(*
SPDX-FileCopyrightText: © 2026 Oleksandr Tiutyk <trofimich@gmail.com>
SPDX-License-Identifier: MIT
License: https://opensource.org/license/mit
*)

(*!
<summary>Reports a rejected filesystem path and its diagnostic explanation.</summary>
<description>
Reports caller-detected path errors using the GeneralException lifetime and throw rules. The path is borrowed
during the call; errorMessage is copied by value. Dynamic copies are explicitly registered by Clone after
construction; plain __NEW does not transfer ownership to the task manager.
</description>
*)

{attribute 'enable_dynamic_creation'}
{attribute 'no_explicit_call' := 'do not call this function block directly'}
FUNCTION_BLOCK InvalidPathException EXTENDS TOF_Core.GeneralException IMPLEMENTS IInvalidPathException
VAR_STAT
	//! <summary>Class name shared by all instances of this function block.</summary>
	{attribute 'hide'} 
	_ClassName : STRING := __POUNAME();
END_VAR

(*!
<summary>Provides the concrete type name used in diagnostics.</summary>
<description>
Returns borrowed read-only metadata; keep the instance alive and do not modify the referenced string.
Reading does not allocate memory, initialize resources or transfer ownership.
</description>
*)
{attribute 'monitoring' := 'call'}
PROPERTY ClassName : REFERENCE TO STRING
GET
ClassName REF= _ClassName;
END_GET
END_PROPERTY

(*!
<summary>Creates a task-owned copy of this exception and its diagnostic payload.</summary>
<description>
Registers the newly constructed instance before copying payload, outside FB_init. Registration failure
releases the unregistered instance and raises a terminal error; copy failure leaves the registered instance
owned by the task manager for cleanup. Custom overrides must follow the same ownership sequence. The returned
reference is borrowed until task cleanup and must not be deleted by the caller.
</description>
*)
METHOD Clone : TOF_Core.IObject
VAR
	exceptionClone : POINTER TO InvalidPathException;
END_VAR
exceptionClone := __NEW(InvalidPathException);

IF exceptionClone = 0 THEN
	TOF_Core.DynamicMemoryManager.RaiseAllocationFailure();
END_IF

TOF_Core.DynamicMemoryManager.RegisterAutoDisposedObject(autoDisposedObject := exceptionClone^);

exceptionClone^.CopyGeneralFields(sourceException := THIS^);

Clone := exceptionClone^;
END_METHOD

(*!
<summary>Provides the library namespace used in diagnostics.</summary>
<description>Returns borrowed read-only namespace storage; do not modify the referenced string.</description>
*)
{attribute 'monitoring' := 'call'}
PROPERTY NamespaceName : REFERENCE TO STRING
GET
NamespaceName REF= CurrentNamespace.Name;
END_GET
END_PROPERTY

(*!
<summary>Reports the size of this concrete instance in bytes.</summary>
*)
{attribute 'monitoring' := 'call'}
PROPERTY SelfSize : ULINT
GET
SelfSize := XSIZEOF(THIS^);
END_GET
END_PROPERTY

(*!
<summary>Raises an exception describing the rejected path and its reason.</summary>
<description>
Borrows path read-only for this call and copies errorMessage by value, limited to 255 characters. Formats
diagnostic text without heap allocation during message preparation; does not retain the input reference. The
caller detects the invalid path; this method does not validate it.
</description>
*)
METHOD Throw
VAR_INPUT
	sourceNamespaceName : STRING;
	sourceClassName : STRING;
	sourcePOUName : STRING;
	sourcePosition : STRING;
END_VAR
VAR_IN_OUT CONSTANT
	path : STRING(255);
END_VAR
VAR_INPUT
	errorMessage : WSTRING(255);
END_VAR
VAR
	message : TOF_Core.ERROR_MESSAGE;
END_VAR
TOF_Core.WideStrings.Append255(
	message,
	"Invalid path ",
	TO_WSTRING('$22'),
	TO_WSTRING(path),
	TO_WSTRING('$22: '),
	errorMessage);

InternalThrow(
	sourceNamespaceName := sourceNamespaceName,
	sourceClassName := sourceClassName,
	sourcePOUName := sourcePOUName,
	sourcePosition := sourcePosition,
	message := message,
	errorCode := 0,
	innerException := 0
);
END_METHOD

END_FUNCTION_BLOCK

(* stored: Version 1.1.0.1
   POU InvalidPathException: Id {548744c4-a8a9-4007-b2c1-225cf445257a}, SpecialFunc None
   Property ClassName: Id {6d3da3bd-a6e5-45c1-bda2-e3e02c19b687}
   Get Get: Id {266b1451-a7f7-4677-9a17-074c37418502}
   Method Clone: Id {bd9b6470-1f00-427e-b60b-49934c91d8f4}
   Property NamespaceName: Id {40a5cc6f-fd53-4b14-9f42-0450d3eda511}
   Get Get: Id {10e0e80e-3bc6-4cdb-a3c8-368be4e2bfe9}
   Property SelfSize: Id {63d69ff8-6f79-48c9-ace4-f2c04e14a203}
   Get Get: Id {71d83967-5c13-49fa-897c-5f7133252b44}
   Method Throw: Id {d47f41f8-35c7-48fd-869f-e96f29dd4029} *)
